FUNCTION_BLOCK FB_LIMIT_WSTRING (* See FB_LIMIT_ANY *)
  (* Standard: IEC 61499 *)
  (* Version 0.1, 2005-06-01, JHC, Holobloc Inc, Moved to fb.rt.strings. *)
  (* Version 0.0, 2004-12-15, JHC, Rockwell Automation, Converted from SRC format. *)
  (* Compiler header: package fb.rt.strings; *)
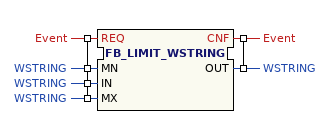
  EVENT_INPUT
    REQ WITH MN, IN, MX;
  END_EVENT
  EVENT_OUTPUT
    CNF WITH OUT;
  END_EVENT
  VAR_INPUT
    MN : WSTRING;
    IN : WSTRING;
    MX : WSTRING;
  END_VAR
  VAR_OUTPUT
    OUT : WSTRING;
  END_VAR
END_FUNCTION_BLOCK
